// TIA Portal V20 export
DATA_BLOCK "F-DB_DataToSafety"   // DB121, F_DB
{ S7_Optimized_Access := 'TRUE' }
// stored: AutoNumber false, InstanceOfName DT_DataToSafety, InstanceOfType UDT
"DT_DataToSafety"
   // VAR
   //    OpenShutterButton : Bool;
   //    ResetEmergencyStop : Bool;
   //    JOG_Mod : Bool;
   //    Activation_Axis : Bool;
   //    CloseShutter : Bool;
   //    FrontDoorLock : Bool;
   //    DoorsInhibit : Bool;
   // END_VAR
BEGIN
END_DATA_BLOCK
